SUBAPPLICATION Uebung_051 (* DigitalInput_I1-_I4 auf DigitalOutput_Q1-_Q4 *)
  (* Standard: 61499-2; Description: Copyright (c) 2023 Meisterschulen am Ostbahnhof This program and the accompanying materials are made available under the terms of the Eclipse Public License 2.0 which is available at https://www.eclipse.org/legal/epl-2.0/ SPDX-License-Identifier: EPL-2.0 *)
  (* Version 1.0, 2023-10-23, Franz Höpfinger, Meisterschulen am Ostbahnhof *)
  IMPORT logiBUS::io::DI::logiBUS_DI::Input_I1;
  IMPORT logiBUS::io::DI::logiBUS_DI::Input_I2;
  IMPORT logiBUS::io::DI::logiBUS_DI::Input_I3;
  IMPORT logiBUS::io::DI::logiBUS_DI::Input_I4;
  IMPORT logiBUS::io::DQ::logiBUS_DO::Output_Q1;
  IMPORT logiBUS::io::DQ::logiBUS_DO::Output_Q2;
  IMPORT logiBUS::io::DQ::logiBUS_DO::Output_Q3;
  IMPORT logiBUS::io::DQ::logiBUS_DO::Output_Q4;
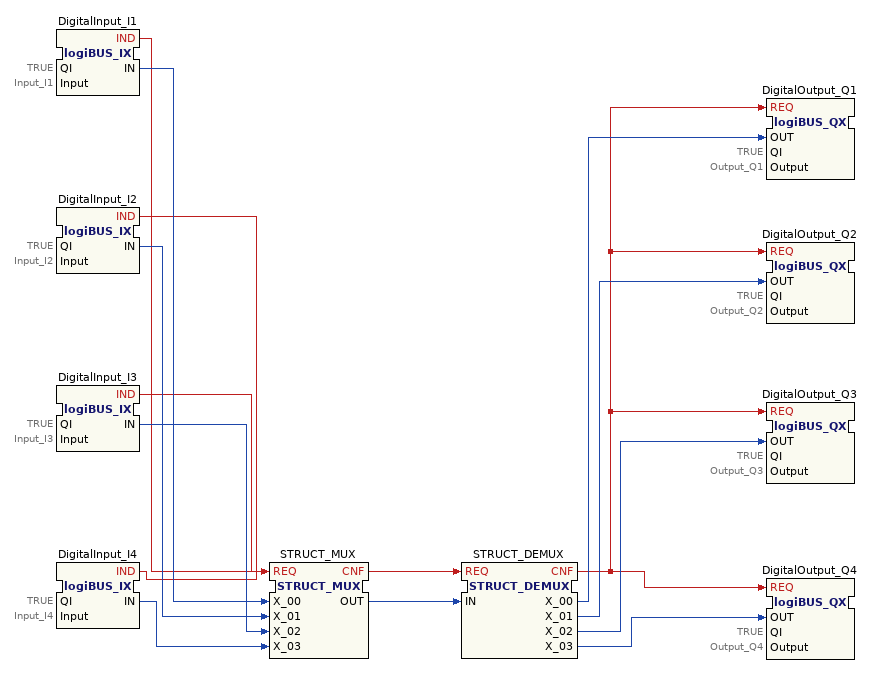
  FBS
    DigitalOutput_Q1 : logiBUS::io::DQ::logiBUS_QX(QI := TRUE, Output := Output_Q1);
    DigitalInput_I1 : logiBUS::io::DI::logiBUS_IX(QI := TRUE, Input := Input_I1);
    DigitalOutput_Q2 : logiBUS::io::DQ::logiBUS_QX(QI := TRUE, Output := Output_Q2);
    DigitalInput_I2 : logiBUS::io::DI::logiBUS_IX(QI := TRUE, Input := Input_I2);
    DigitalOutput_Q3 : logiBUS::io::DQ::logiBUS_QX(QI := TRUE, Output := Output_Q3);
    DigitalInput_I3 : logiBUS::io::DI::logiBUS_IX(QI := TRUE, Input := Input_I3);
    DigitalOutput_Q4 : logiBUS::io::DQ::logiBUS_QX(QI := TRUE, Output := Output_Q4);
    DigitalInput_I4 : logiBUS::io::DI::logiBUS_IX(QI := TRUE, Input := Input_I4);
    STRUCT_DEMUX : eclipse4diac::convert::STRUCT_DEMUX; {SET_ATTRIBUTE(StructuredType, logiBUS::utils::conversion::types::ST04X)}
    STRUCT_MUX : eclipse4diac::convert::STRUCT_MUX; {SET_ATTRIBUTE(StructuredType, logiBUS::utils::conversion::types::ST04X)}
  END_FBS
  EVENT_CONNECTIONS
    DigitalInput_I1.IND TO STRUCT_MUX.REQ;
    DigitalInput_I2.IND TO STRUCT_MUX.REQ;
    DigitalInput_I3.IND TO STRUCT_MUX.REQ;
    DigitalInput_I4.IND TO STRUCT_MUX.REQ;
    STRUCT_MUX.CNF TO STRUCT_DEMUX.REQ;
    STRUCT_DEMUX.CNF TO DigitalOutput_Q1.REQ;
    STRUCT_DEMUX.CNF TO DigitalOutput_Q2.REQ;
    STRUCT_DEMUX.CNF TO DigitalOutput_Q3.REQ;
    STRUCT_DEMUX.CNF TO DigitalOutput_Q4.REQ;
  END_CONNECTIONS
  DATA_CONNECTIONS
    DigitalInput_I1.IN TO STRUCT_MUX.X_00;
    DigitalInput_I2.IN TO STRUCT_MUX.X_01;
    DigitalInput_I3.IN TO STRUCT_MUX.X_02;
    DigitalInput_I4.IN TO STRUCT_MUX.X_03;
    STRUCT_MUX.OUT TO STRUCT_DEMUX.IN;
    STRUCT_DEMUX.X_00 TO DigitalOutput_Q1.OUT;
    STRUCT_DEMUX.X_01 TO DigitalOutput_Q2.OUT;
    STRUCT_DEMUX.X_02 TO DigitalOutput_Q3.OUT;
    STRUCT_DEMUX.X_03 TO DigitalOutput_Q4.OUT;
  END_CONNECTIONS
END_SUBAPPLICATION
